// TIA Portal V19 export
TYPE "HU_Pump_HMI"
// stored: Access Published
   STRUCT
      Alarm : Bool;
      ManStart : Bool;
      PumpRunning : Bool;
      PressureRunning : Bool;
   END_STRUCT;
END_TYPE
